{attribute 'qualified_only'}
{attribute 'strict'}
TYPE Material_Type :
(
	Plastic := 0,
	Metal :=1
);
END_TYPE

(* stored: Version 1.1.0.1, ProductVersion 3.1.4024.3
   DUT Material_Type: Id {04893429-dd74-43e0-aa26-a7440767e584} *)
